(* IEC 61131-3 sources: volt/packages/volt-lsp-iec/test-corpus/lenze-mid/Device/Plc Logic/Application/Library Manager/SysSem Implementation, 5 files *)

(* ---- SYSSEMCREATE.pou ---- *)
FUNCTION SYSSEMCREATE : RTS_IEC_HANDLE
VAR_INPUT
	PRESULT : POINTER TO RTS_IEC_RESULT;
END_VAR
END_FUNCTION

(* ---- SYSSEMDELETE.pou ---- *)
FUNCTION SYSSEMDELETE : RTS_IEC_RESULT
VAR_INPUT
	HSEM : RTS_IEC_HANDLE;
END_VAR
END_FUNCTION

(* ---- SYSSEMENTER.pou ---- *)
FUNCTION SYSSEMENTER : RTS_IEC_RESULT
VAR_INPUT
	HSEM : RTS_IEC_HANDLE;
END_VAR
END_FUNCTION

(* ---- SYSSEMLEAVE.pou ---- *)
FUNCTION SYSSEMLEAVE : RTS_IEC_RESULT
VAR_INPUT
	HSEM : RTS_IEC_HANDLE;
END_VAR
END_FUNCTION

(* ---- SYSSEMTRY.pou ---- *)
FUNCTION SYSSEMTRY : RTS_IEC_RESULT
VAR_INPUT
	HSEM : RTS_IEC_HANDLE;
END_VAR
END_FUNCTION
